FUNCTION_BLOCK Faults2
VAR_INPUT
END_VAR
VAR_OUTPUT
END_VAR
VAR
END_VAR

END_FUNCTION_BLOCK

(* stored: Version 1.1.0.1, ProductVersion 3.1.4024.11
   POU Faults2: Id {48406e60-56d9-479c-aae9-1deb43b91d18}, SpecialFunc None *)
